{attribute 'qualified_only'}
VAR_GLOBAL
	sPistonEndStopMessage : STRING;
END_VAR

(* stored: Version 1.1.0.1, ProductVersion 3.1.4024.10
   GVL HMI: Id {181c680c-2292-4a10-ba52-8c49ff7b85ed} *)
